{attribute 'linkalways'}
{attribute 'no_explicit_call' := 'This FB is a CLASS and must be accessed using methods or properties'}
{attribute 'enable_dynamic_creation'}
FUNCTION_BLOCK Node_F_VN_AnalyzeBarcodeWalsh EXTENDS VisionNode
VAR
    ipBarcodeImage : _ITcVnImage;
    stParams : _TcVnParamsWalshBarcodeDetection;
    hrPrev : _HRESULT(S_OK);
    hresult : _HRESULT(S_OK);
END_VAR

METHOD PUBLIC Clone : I_Node
VAR
    pNode : POINTER TO Node_F_VN_AnalyzeBarcodeWalsh;
END_VAR
pNode := __NEW(Node_F_VN_AnalyzeBarcodeWalsh);
Clone := pNode^;
END_METHOD

METHOD FB_init : BOOL
VAR_INPUT
    bInitRetains : BOOL;
    bInCopyCode : BOOL;
END_VAR
AddInput('ipBarcodeImage', ipBarcodeImage);
AddInput('stParams', stParams);
AddInput('hrPrev', hrPrev);
AddOutput('stParams', stParams);
AddOutput('hresult', hresult);
END_METHOD

METHOD PROTECTED OnExecute
hresult.Value := F_VN_AnalyzeBarcodeWalsh(
    ipBarcodeImage := ipBarcodeImage.Value,
    stParams := stParams.Value,
    hrPrev := hrPrev.Value);
END_METHOD

METHOD PUBLIC PreExecutionCheck
VAR_INPUT
    Check : I_PreExecutionChecks;
END_VAR
Check.IsTrue(ipBarcodeImage.IsValid, 'ipBarcodeImage must contain an image');
END_METHOD

END_FUNCTION_BLOCK

(* stored: Version 1.1.0.1, ProductVersion 3.1.4026.19
   POU Node_F_VN_AnalyzeBarcodeWalsh: Id {c607d63a-2fa0-44c2-be62-23875eb150c5}, SpecialFunc None
   Folder Constructor: Id {d5743ad7-1f0e-4828-9f02-042bbf5aacce}
   Method Clone: Id {44e29a3e-edeb-4358-b81e-35370ba4e559}
   Method FB_init: Id {69f15610-6671-4cf1-a5e6-bc8f10f5b0c1}
   Method OnExecute: Id {eb7e3c59-9659-4ff7-ae6e-b5e2dc566e61}
   Method PreExecutionCheck: Id {007dc5eb-6d04-4eca-8c75-5e0e145f397a} *)
